INTERFACE I_ValveIo EXTENDS I_Device

METHOD M_ManualControl : BOOL
VAR_INPUT
	ManualTrigValve : ARRAY[0..31] OF BOOL;
END_VAR
END_METHOD

METHOD M_MapMaskToOutBytes
VAR_INPUT
END_VAR
END_METHOD

METHOD M_ValvePositionOK : BOOL
VAR_INPUT
END_VAR
END_METHOD

PROPERTY pNumOfChannels : INT
GET
END_GET
SET
END_SET
END_PROPERTY

PROPERTY pNumOfValvesAvailable : INT
GET
END_GET
SET
END_SET
END_PROPERTY

PROPERTY pValveMaskInput : DWORD
SET
END_SET
END_PROPERTY

PROPERTY pValveMaskOutBYTE : ARRAY[0..3] OF BYTE
GET
END_GET
END_PROPERTY

PROPERTY pValveMaskOutDINT : DINT
GET
END_GET
END_PROPERTY

PROPERTY pValveMaskOutDWORD : DWORD
GET
END_GET
END_PROPERTY

PROPERTY pValveMaskOutINT : ARRAY[0..1] OF INT
GET
END_GET
END_PROPERTY

PROPERTY pValveMaskOutSINT : ARRAY[0..3] OF SINT
GET
END_GET
END_PROPERTY

PROPERTY pValveMaskOutWORD : ARRAY[0..1] OF WORD
GET
END_GET
END_PROPERTY

PROPERTY pValvePositionFeedback : DWORD
SET
END_SET
END_PROPERTY

END_INTERFACE

(* stored: Version 1.1.0.1
   Itf I_ValveIo: Id {9abff4a5-9dc4-4338-a357-8d967cc6368b}
   Method M_ManualControl: Id {63fac6b4-9286-4ff2-830b-5a885f2ba6a0}
   Method M_MapMaskToOutBytes: Id {755f9910-c101-4fb7-90ee-bcba44a6a4a3}
   Method M_ValvePositionOK: Id {a1eac1b7-3181-4ced-9150-59d0318060bd}
   Property pNumOfChannels: Id {e2f540e3-a647-4887-b05a-79e0b0c456f7}
   Get Get: Id {e67456f8-dd4a-4c5e-ab39-b721f030e82f}
   Set Set: Id {b48f9988-9810-4cc2-b8f1-1c3d55fe87ae}
   Property pNumOfValvesAvailable: Id {f7ac2a41-ab7b-4416-8cf9-6ea4b760921c}
   Get Get: Id {1fb65154-0e04-4899-90af-8f762ad2b37c}
   Set Set: Id {f59aaf3d-2dea-4a6d-9e63-928ca745b81c}
   Property pValveMaskInput: Id {a2bf4f17-8acc-4c24-9eb3-27d4979bba01}
   Set Set: Id {0cd549e6-c2c7-4c72-bc8b-00d6685b8fd8}
   Property pValveMaskOutBYTE: Id {1ee32bb6-fd44-4bb7-94af-44c409f2bc06}
   Get Get: Id {3f2a80d1-2a49-447a-8947-7db9a1c75cf2}
   Property pValveMaskOutDINT: Id {cfaea788-7599-476d-9bc2-31b81c3bc89c}
   Get Get: Id {843e320a-605f-48a1-a25a-6faceccb9cc5}
   Property pValveMaskOutDWORD: Id {ac7ba397-3b3b-4a5c-acc8-c7f7d62d2ed3}
   Get Get: Id {37006514-9632-4a5d-bb42-7ec39080674d}
   Property pValveMaskOutINT: Id {0907e569-f36c-4bcb-b139-f461796d20c3}
   Get Get: Id {59cf7d33-61bd-4b00-85a6-881a8718f31c}
   Property pValveMaskOutSINT: Id {ea11584c-ad6f-4276-bf76-f031e87e0e90}
   Get Get: Id {7ab9c677-32a9-4418-90ad-4ce8ab205e3e}
   Property pValveMaskOutWORD: Id {02b1fa7a-6aea-45ae-bfb8-803a72216ab7}
   Get Get: Id {2c0e895e-7086-4d0e-8430-60874d40d872}
   Property pValvePositionFeedback: Id {c55bfe97-8d3b-45da-a426-2abf1a4d9ef0}
   Set Set: Id {084da671-2287-4f87-9230-3828fc2a8438} *)
